KUKA KRL data list: LAB_MISSING_TARGET.dat

&ACCESS RVP
&REL 1
DEFDAT LAB_MISSING_TARGET PUBLIC
  DECL E6AXIS A_HOME={A1 0,A2 -90,A3 90,A4 0,A5 0,A6 0,E1 0,E2 0,E3 0,E4 0,E5 0,E6 0}
ENDDAT
